// TIA Portal V17 export
// export: Created 2021-11-12T21:16:16.4740391Z, ExportSetting WithDefaults, DisplayName Totally Integrated Automation Portal, DisplayVersion V17 Update 1, DisplayName TIA Portal Openness, DisplayVersion V17 Update 1, DisplayName TIA Portal Version Control Interface, DisplayVersion V17, DisplayName SINAMICS Startdrive Advanced, DisplayVersion V17 Update1, DisplayName SINAMICS Startdrive G110M, G120, G120C, G120D, G120P, G115D, DisplayVersion V17 Update1, DisplayName SINAMICS Startdrive G130, G150, S120, S150, SINAMICS MV, S210, DisplayVersion V17 Update1, DisplayName STEP 7 Professional, DisplayVersion V17 Update 1, DisplayName STEP 7 Safety, DisplayVersion V17, DisplayName WinCC Advanced, DisplayVersion V17 Update 1
VAR_GLOBAL   // PLC tag table "Default tag table"
   System_Byte AT %MB100 : Byte;
   FirstScan AT %M100.0 : Bool;
   DiagStatusUpdate AT %M100.1 : Bool;
   AlwaysTRUE AT %M100.2 : Bool;
   AlwaysFALSE AT %M100.3 : Bool;
   Clock_Byte AT %MB101 : Byte;
   Clock_10Hz AT %M101.0 : Bool;
   Clock_5Hz AT %M101.1 : Bool;
   "Clock_2.5Hz" AT %M101.2 : Bool;
   Clock_2Hz AT %M101.3 : Bool;
   "Clock_1.25Hz" AT %M101.4 : Bool;
   Clock_1Hz AT %M101.5 : Bool;
   "Clock_0.625Hz" AT %M101.6 : Bool;
   "Clock_0.5Hz" AT %M101.7 : Bool;
   M_CurrentDateTimeStatus AT %MW166 : Int;
END_VAR
